// TIA Portal V15.1 export
// export: Created 2022-12-20T09:13:23.8568367Z, ExportSetting None, DisplayName Totally Integrated Automation Portal, DisplayVersion V15.1 Update 1, DisplayName TIA Portal Openness, DisplayVersion V15.1, DisplayName SINAMICS Startdrive Advanced, DisplayVersion V15.1, DisplayName G130, G150, S120, S150, SINAMICS MV, S210, DisplayVersion V15.1, DisplayName G110M, G120, G120C, G120D, G120P, DisplayVersion V15.1, DisplayName STEP 7 Professional, DisplayVersion V15.1 Update 1, DisplayName STEP 7 Safety, DisplayVersion V15.1, DisplayName WinCC Professional, DisplayVersion V15.1 Update 1, DisplayName SIMATIC Visualization Architect, DisplayVersion V15.1
FUNCTION_BLOCK "PLC_Type_FB"   // FB514, FBD
TITLE = PLC_TYPE_FB
{ S7_Optimized_Access := 'FALSE' }
// The block is used to control main type fb
// stored: AutoNumber false, SetENOAutomatically False
   VAR
      Type_Buffer : "Type_Buffer_FB";   // Type buffer
      Type_Manager : "Type_Manager_FB";   // Memory Locations for process status used, and references active
   END_VAR
BEGIN

REGION Network 1: Type Manager
   // Memory Locations for process status used, and references active
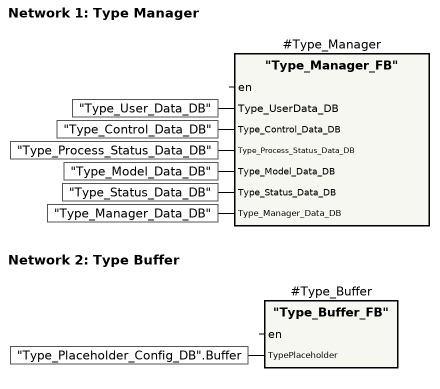
   #Type_Manager(Type_UserData_DB := "Type_User_Data_DB",   // "Type_Manager_FB"
                 Type_Control_Data_DB := "Type_Control_Data_DB",
                 Type_Process_Status_Data_DB := "Type_Process_Status_Data_DB",
                 Type_Model_Data_DB := "Type_Model_Data_DB",
                 Type_Status_Data_DB := "Type_Status_Data_DB",
                 Type_Manager_Data_DB := "Type_Manager_Data_DB");
END_REGION

REGION Network 2: Type Buffer
   // Temporary type placeholder called buffer
   #Type_Buffer(TypePlaceholder := "Type_Placeholder_Config_DB".Buffer);   // "Type_Buffer_FB"
END_REGION
END_FUNCTION_BLOCK
